Universal Robots PolyScope program: wrist_rotate 01.urp

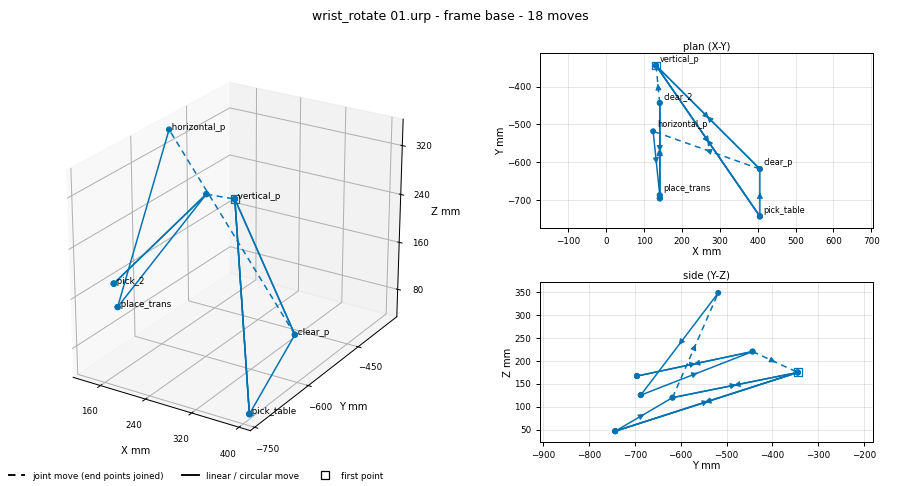
[picture p0: tool path of wrist_rotate 01.urp in frame base, 18 of 19 moves have a stored position in this frame; points joined in program order, loops and branches not executed]
Program wrist_rotate 01 (installation=default directory=/programs createdIn=5.9.1.1031110 lastSavedIn=5.9.1.1031110 robotSerialNumber=20195501059)
Calibrated DH parameters: a=[0.000146, -0.418764, -0.053981, 0.000058, -0.000023, 0]; d=[0.162545, 37.319448, -206.067439, 168.881546, 0.09955, 0.099464]; alpha=[1.57004, -0.001979, 0.002304, 1.570607, -1.57066, 0]; deltaTheta=[0, -0.174616, -1.258233, 1.432844, -0.000001, 0]
BeforeStart
  URCap Gripper Activate (Robotiq_Grippers, Robotiq Inc.) dataModel(ResetAndActivateKey=false)
  start_p := get_actual_tcp_pose()
  MoveJ speed 60 deg/s, acceleration 80 deg/s^2 (useActiveTCP=true) feature=Base
    Waypoint Waypoint (Variable): variable=start_p
Robot Program (runOnlyOnce=true)
  MoveJ speed 60 deg/s, acceleration 80 deg/s^2 (useActiveTCP=true) feature=Base
    Waypoint vertical_p: TCP in base x=131.579 y=-344.603 z=175.048 mm, rx=-2.1692 ry=-2.2724 rz=0 rad; joints [89.678, -107.764, 125.374, -107.601, 270.065, 87.008] deg; TCP offset x=0 y=0 z=174 mm, rx=0 ry=0 rz=0 rad
    URCap Gripper (Robotiq_Grippers, Robotiq Inc.) dataModel(position=100.0, force=100.0, speed=100.0, positionInDouble=100.0, forceInDouble=100.0, speedInDouble=100.0, slaveIds=[9], blocking=true)
  MoveL speed 250 mm/s, acceleration 1200 mm/s^2 (useActiveTCP=true) feature=Base
    Waypoint pick_table: TCP in base x=405.758 y=-742.905 z=46.866 mm, rx=-2.1929 ry=-2.2496 rz=0 rad; joints [109.558, -34.082, 45.933, -101.842, 269.918, 108.061] deg
    MoveDirectionNode (selectedDirection=ZPlus toolParams=0.02, 1.2) feature=Joint_6_name
      Until TOOL_CONTACT_DETECTION (allowActions=true retraction=0.002 decelerationAcceleration=3 decelerationAngularAcceleration=34.906585)
        URCap Gripper (Robotiq_Grippers, Robotiq Inc.) dataModel(position=50.0, force=100.0, speed=100.0, positionInDouble=50.0, forceInDouble=100.0, speedInDouble=100.0, slaveIds=[9], blocking=true)
        MoveDirectionNode (selectedDirection=ZPlus toolParams=0.02, 1.2) feature=Joint_6_name
          Until DISTANCE (allowActions=false deceleration=3 distanceNodeType=STOP) Distance=0.02; motionParameters(blendRadius=0)
        URCap Gripper (Robotiq_Grippers, Robotiq Inc.) dataModel(position=100.0, force=100.0, speed=100.0, positionInDouble=100.0, forceInDouble=100.0, speedInDouble=100.0, slaveIds=[9], blocking=true)
        MoveL speed 250 mm/s, acceleration 1200 mm/s^2 (useActiveTCP=true) feature=Base
          Waypoint pick_table: motionParameters(blendRadius=0.025); TCP in base x=405.758 y=-742.905 z=46.866 mm, rx=-2.1929 ry=-2.2496 rz=0 rad; joints [109.558, -34.082, 45.933, -101.842, 269.918, 108.061] deg
      Until DISTANCE (allowActions=true deceleration=3 distanceNodeType=STOP) Distance=0.02; motionParameters(blendRadius=0)
        Popup Message (haltProgram=false message=part missing inputType=Text)
        MoveL speed 250 mm/s, acceleration 1200 mm/s^2 (useActiveTCP=true) feature=Base
          Waypoint vertical_p: TCP in base x=131.579 y=-344.603 z=175.048 mm, rx=-2.1692 ry=-2.2724 rz=0 rad; joints [89.678, -107.764, 125.374, -107.601, 270.065, 87.008] deg
  MoveL speed 250 mm/s, acceleration 1200 mm/s^2 (useActiveTCP=true) feature=Base
    Waypoint clear_p: TCP in base x=405.743 y=-617.915 z=120.078 mm, rx=-2.1929 ry=-2.2495 rz=0 rad; joints [112.864, -53.763, 70.34, -106.562, 269.959, 111.396] deg
  MoveJ speed 60 deg/s, acceleration 80 deg/s^2 (useActiveTCP=true) feature=Base
    Waypoint horizontal_p: TCP in base x=123.861 y=-518.161 z=348.489 mm, rx=1.214 ry=-1.1859 rz=1.1469 rad; joints [89.68, -107.762, 125.375, -17.506, 91.371, 87.006] deg
  MoveL speed 250 mm/s, acceleration 1200 mm/s^2 (useActiveTCP=true) feature=Base
    Waypoint place_trans: TCP in base x=141.374 y=-687.139 z=125.571 mm, rx=1.2065 ry=-1.18 rz=1.2144 rad; joints [90.758, -63.351, 118.718, -56.546, 90.342, 89.218] deg
    MoveDirectionNode (selectedDirection=ZMinus toolParams=0.01, 1.2)
      Until TOOL_CONTACT_DETECTION (allowActions=true retraction=0 decelerationAcceleration=3 decelerationAngularAcceleration=34.906585)
        URCap Gripper (Robotiq_Grippers, Robotiq Inc.) dataModel(position=50.0, force=100.0, speed=100.0, positionInDouble=50.0, forceInDouble=100.0, speedInDouble=100.0, slaveIds=[9], blocking=true)
    Waypoint place_trans: motionParameters(blendRadius=0.025); TCP in base x=141.374 y=-687.139 z=125.571 mm, rx=1.2065 ry=-1.18 rz=1.2144 rad; joints [90.758, -63.351, 118.718, -56.546, 90.342, 89.218] deg
    Waypoint clear_2: TCP in base x=141.36 y=-443.257 z=220.65 mm, rx=1.5969 ry=-1.558 rz=0.9277 rad; joints [90.999, -105.53, 124.958, 9.942, 89.916, 89.647] deg
  MoveL speed 250 mm/s, acceleration 1200 mm/s^2 (useActiveTCP=true) feature=Base
    URCap Gripper (Robotiq_Grippers, Robotiq Inc.) dataModel(position=100.0, force=100.0, speed=100.0, positionInDouble=100.0, forceInDouble=100.0, speedInDouble=100.0, slaveIds=[9], blocking=true)
    Waypoint pick_2: TCP in base x=141.376 y=-695.44 z=167.162 mm, rx=1.2065 ry=-1.1801 rz=1.2144 rad; joints [90.745, -67.554, 116.133, -49.758, 90.319, 89.221] deg
    MoveDirectionNode (selectedDirection=ZMinus toolParams=0.02, 1.2) feature=Base
      Until DISTANCE (allowActions=true deceleration=3 distanceNodeType=STOP) Distance=0.02; motionParameters(blendRadius=0)
        Popup Message (haltProgram=false message=part_missing inputType=Text)
        MoveL speed 250 mm/s, acceleration 1200 mm/s^2 (useActiveTCP=true) feature=Base
          Waypoint pick_2: TCP in base x=141.376 y=-695.44 z=167.162 mm, rx=1.2065 ry=-1.1801 rz=1.2144 rad; joints [90.745, -67.554, 116.133, -49.758, 90.319, 89.221] deg
      Until TOOL_CONTACT_DETECTION (allowActions=true retraction=0.001 decelerationAcceleration=3 decelerationAngularAcceleration=34.906585)
        URCap Gripper (Robotiq_Grippers, Robotiq Inc.) dataModel(position=50.0, force=100.0, speed=100.0, positionInDouble=50.0, forceInDouble=100.0, speedInDouble=100.0, slaveIds=[9], blocking=true)
        MoveDirectionNode (selectedDirection=ZMinus toolParams=0.03, 1.2) feature=Base
          Until DISTANCE (allowActions=false deceleration=3 distanceNodeType=STOP) Distance=0.035; motionParameters(blendRadius=0)
        URCap Gripper (Robotiq_Grippers, Robotiq Inc.) dataModel(position=100.0, force=100.0, speed=100.0, positionInDouble=100.0, forceInDouble=100.0, speedInDouble=100.0, slaveIds=[9], blocking=true)
    Waypoint pick_2: TCP in base x=141.376 y=-695.44 z=167.162 mm, rx=1.2065 ry=-1.1801 rz=1.2144 rad; joints [90.745, -67.554, 116.133, -49.758, 90.319, 89.221] deg
    Waypoint clear_2: TCP in base x=141.36 y=-443.257 z=220.65 mm, rx=1.5969 ry=-1.558 rz=0.9277 rad; joints [90.999, -105.53, 124.958, 9.942, 89.916, 89.647] deg
  MoveJ speed 60 deg/s, acceleration 80 deg/s^2 (useActiveTCP=true) feature=Base
    Waypoint vertical_p: TCP in base x=131.579 y=-344.603 z=175.048 mm, rx=-2.1692 ry=-2.2724 rz=0 rad; joints [89.678, -107.764, 125.374, -107.601, 270.065, 87.008] deg
  MoveL speed 250 mm/s, acceleration 1200 mm/s^2 (useActiveTCP=true) feature=Base
    Waypoint pick_table: TCP in base x=405.758 y=-742.905 z=46.866 mm, rx=-2.1929 ry=-2.2496 rz=0 rad; joints [109.558, -34.082, 45.933, -101.842, 269.918, 108.061] deg
    MoveDirectionNode (selectedDirection=ZMinus toolParams=0.02, 1.2) feature=Base
      Until TOOL_CONTACT_DETECTION (allowActions=true retraction=0 decelerationAcceleration=3 decelerationAngularAcceleration=34.906585)
        URCap Gripper (Robotiq_Grippers, Robotiq Inc.) dataModel(position=50.0, force=100.0, speed=100.0, positionInDouble=50.0, forceInDouble=100.0, speedInDouble=100.0, slaveIds=[9], blocking=true)
        Waypoint pick_table: TCP in base x=405.758 y=-742.905 z=46.866 mm, rx=-2.1929 ry=-2.2496 rz=0 rad; joints [109.558, -34.082, 45.933, -101.842, 269.918, 108.061] deg
        Waypoint clear_p: motionParameters(blendRadius=0.025); TCP in base x=405.743 y=-617.915 z=120.078 mm, rx=-2.1929 ry=-2.2495 rz=0 rad; joints [112.864, -53.763, 70.34, -106.562, 269.959, 111.396] deg
        Waypoint vertical_p: TCP in base x=131.579 y=-344.603 z=175.048 mm, rx=-2.1692 ry=-2.2724 rz=0 rad; joints [89.678, -107.764, 125.374, -107.601, 270.065, 87.008] deg
